FUNCTION_BLOCK Motor_VFD
VAR_INPUT
	//Run Feedback from Motor Starter
	Run_Feedback : BOOL; 
	//Reset trigger for Runtime Maint
	Runtime_Maint_Reset : BOOL;
	//Run Request from PLC Program
	Run_Request : BOOL;
	//Requested Speed From PLC Program
	Speed_Request : REAL;
	//Speed Feedback from VFD
	Speed_Feedback : REAL;
	//VFD Fault Status from VFD
	VFD_Fault : BOOL;
	//True if Run Command is true and Run Feedback is false for 3 seconds
	Fail_to_Start : BOOL;
	//True if Run Command is false and Run Feedback is true for 3 seconds
	Fail_to_Stop : BOOL;
	//Daily Reset from GENERAL POU
	Daily_Reset : BOOL;
END_VAR
VAR_OUTPUT
	//Tells the motor to start when true, stop when false
	Run_Command : BOOL;
	//VFD Fault Alarm
	Runtime_Today : REAL;
	//Accumulated Runtime Hours Today
	Runtime_Total : REAL;
	//Resettable Runtime for Maintenance purposes, Description is user adjustable
	Runtime_Maint : REAL;
	//Speed Command to VFD
	Speed_Command : REAL;
END_VAR
VAR
	//Runtime Timer Tags, 1 Minute Timer
	Runtime_TON : TON;
	Runtime_PT : TIME := T#1M;
	Runtime_ET : TIME;
	//Runtime Today Counter
	Runtime_Today_CTU : CTU;
	Runtime_Today_CTU_PV : WORD;
	Runtime_Today_CTU_CV : REAL;
	//Total Runtime Minute Counter
	Runtime_Total_Minute_CTU : CTU;
	Runtime_Total_Minute_CTU_Reset : BOOL;
	Runtime_Total_Minute_CTU_PV : WORD :=60;
	Runtime_Total_Minute_CTU_CV : REAL;
	//Total Runtime Hour Counter
	Runtime_Total_Hour_CTU : CTU;
	Runtime_Total_Hour_CTU_Reset : BOOL;
	Runtime_Total_Hour_CTU_PV : WORD;
	//Maintenance Runtime Minute Counter
	Runtime_Maint_Minute_CTU : CTU;
	Runtime_Maint_Minute_CTU_Reset : BOOL;
	Runtime_Maint_Minute_CTU_PV : WORD :=60;
	Runtime_Maint_Minute_CTU_CV : REAL;
	//Maintenance Runtime Hour Counter
	Runtime_Maint_Hour_CTU : CTU;
	Runtime_Maint_Hour_CTU_PV : WORD;
END_VAR
VAR // added by the converter: edge detectors and wires of the graphical bodies
    _w1, _w2 : BOOL;
END_VAR

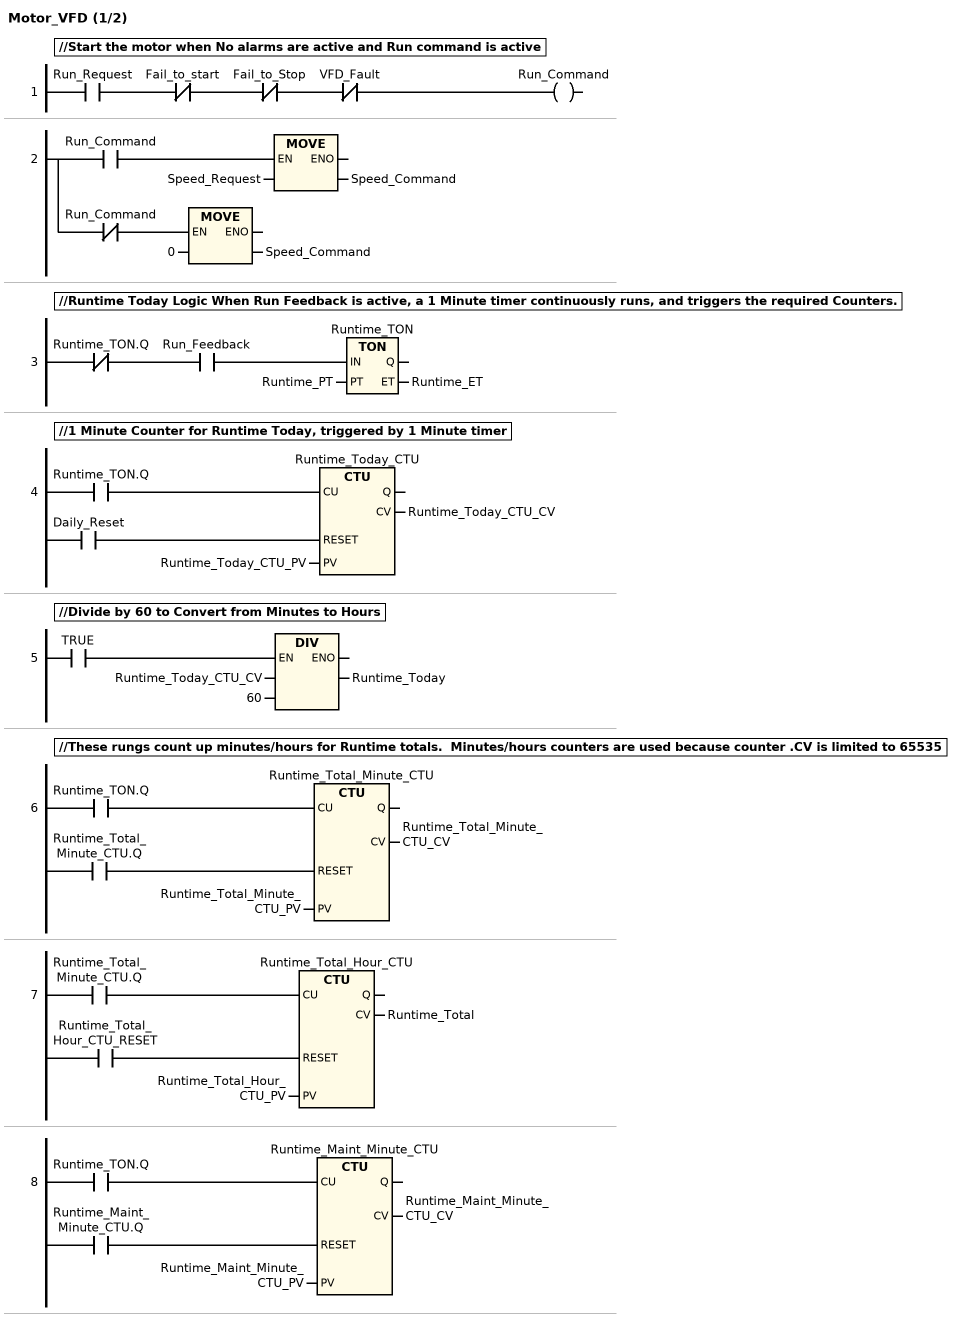
// NETWORK 1
// label: //Start the motor when No alarms are active and Run command is active
Run_Command := Run_Request AND NOT Fail_to_start AND NOT Fail_to_Stop AND NOT VFD_Fault;

// NETWORK 2
_w1 := Run_Command;
IF _w1 THEN Speed_Command := Speed_Request; END_IF
_w2 := NOT Run_Command;
IF _w2 THEN Speed_Command := 0; END_IF
(* _w1 OR _w2; result not used *)

// NETWORK 3
// label: //Runtime Today Logic When Run Feedback is active, a 1 Minute timer continuously runs, and triggers the required Counters.
Runtime_TON(IN := NOT Runtime_TON.Q AND Run_Feedback, PT := Runtime_PT, ET => Runtime_ET); // TON

// NETWORK 4
// label: //1 Minute Counter for Runtime Today, triggered by 1 Minute timer
Runtime_Today_CTU(
    CU := Runtime_TON.Q,
    RESET := Daily_Reset,
    PV := Runtime_Today_CTU_PV,
    CV => Runtime_Today_CTU_CV); // CTU

// NETWORK 5
// label: //Divide by 60 to Convert from Minutes to Hours
Runtime_Today := Runtime_Today_CTU_CV / 60;

// NETWORK 6
// label: //These rungs count up minutes/hours for Runtime totals.  Minutes/hours counters are used because counter .CV is limited to 65535
Runtime_Total_Minute_CTU(
    CU := Runtime_TON.Q,
    RESET := Runtime_Total_Minute_CTU.Q,
    PV := Runtime_Total_Minute_CTU_PV,
    CV => Runtime_Total_Minute_CTU_CV); // CTU

// NETWORK 7
Runtime_Total_Hour_CTU(
    CU := Runtime_Total_Minute_CTU.Q,
    RESET := Runtime_Total_Hour_CTU_RESET,
    PV := Runtime_Total_Hour_CTU_PV,
    CV => Runtime_Total); // CTU

// NETWORK 8
Runtime_Maint_Minute_CTU(
    CU := Runtime_TON.Q,
    RESET := Runtime_Maint_Minute_CTU.Q,
    PV := Runtime_Maint_Minute_CTU_PV,
    CV => Runtime_Maint_Minute_CTU_CV); // CTU

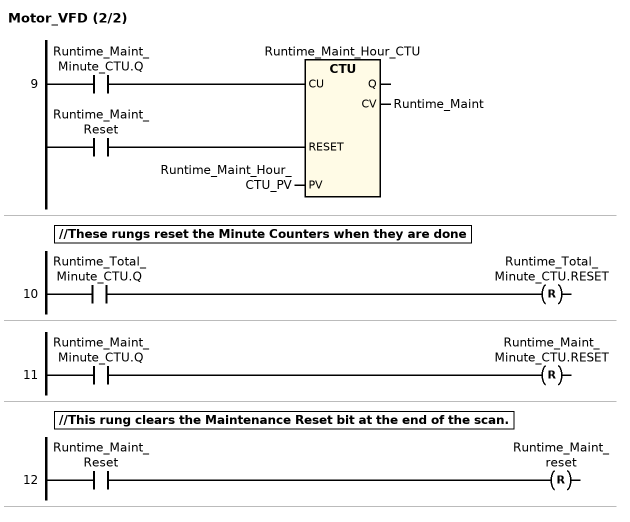
// NETWORK 9
Runtime_Maint_Hour_CTU(
    CU := Runtime_Maint_Minute_CTU.Q,
    RESET := Runtime_Maint_Reset,
    PV := Runtime_Maint_Hour_CTU_PV,
    CV => Runtime_Maint); // CTU

// NETWORK 10
// label: //These rungs reset the Minute Counters when they are done
Runtime_Total_Minute_CTU.RESET R= Runtime_Total_Minute_CTU.Q;

// NETWORK 11
Runtime_Maint_Minute_CTU.RESET R= Runtime_Maint_Minute_CTU.Q;

// NETWORK 12
// label: //This rung clears the Maintenance Reset bit at the end of the scan.
Runtime_Maint_reset R= Runtime_Maint_Reset;

END_FUNCTION_BLOCK

(* stored: Version 1.1.0.1, ProductVersion 3.1.4024.12
   POU Motor_VFD: Id {60a210a4-48dd-4db3-b672-c8198b95c310}, SpecialFunc None *)
